# EPICS StreamDevice protocol: IOC/ArduinoIOC/ArduinoIOCApp/Db/arduino.proto
Terminator = LF;
get_analog {
	out "R";
	in "R %f";
	ExtraInput = Ignore;
}
set_digital {
	out "W%d";
	ExtraInput = Ignore;
}
